Omron Sysmac Studio project testbed_1 (Sysmac Studio 1.30.0.17, StandardProject)

# Controller testbed_1: NX102-1000 version 1.40
Units and slaves: Unit 1 : NX-ECS112 (N1); Unit 2 : NX-PF0730 (N2); Unit 3 : NX-OD5256 (N3); Unit 4 : NX-ID5442 (N4); Unit 5 : NX-AD2604 (N5)
Axis Ax_Servo, settings changed from default: AxisType=ServoType, UnitsConversion=EnumElement5, UnitsNumerator=8388608, ReducerUse=EnumElement2, UnitsDenominator=360, TravelDistancePerWorkRotation=360, MotorGearRatio=30, MaxVelocity=600, MaxJogVelocity=90, InPositionBand=0.1, ZeroPositionBand=0.1, SoftwareLimitMode=ValidForSpecifiedValueDecreaseStop, PositiveSoftwareLimit=91, NegativeSoftwareLimit=-91, HomingVelocity=10, HomingApproachVelocity=10, CompensationVelocity=10, ModuloMAXPosition=180, ModuloMINPosition=-180
Axis Ax_Pendulum, settings changed from default: AxisNumber=1, AxisType=EncoderType, UnitsConversion=EnumElement5, UnitsNumerator=16384, UnitsDenominator=360, ActualVelocityFilterTime=100, CountMode=EnumElement2, ModuloMAXPosition=180, ModuloMINPosition=-180, EncoderTypes=Abs
Task PrimaryTask (priority 4, period or condition 1000): main

VAR_GLOBAL
    N1_Ch1_Encoder_Present_Position : DINT;  (* at IOBus://unit#1/Ch1 Encoder Present Position *)
    N3_Output_Bit_00 : BOOL;  (* at IOBus://unit#3/Output Bit 16 bits/Output Bit 00 *)
    N3_Output_Bit_01 : BOOL;  (* at IOBus://unit#3/Output Bit 16 bits/Output Bit 01 *)
    N3_Output_Bit_02 : BOOL;  (* at IOBus://unit#3/Output Bit 16 bits/Output Bit 02 *)
    N3_Output_Bit_03 : BOOL;  (* at IOBus://unit#3/Output Bit 16 bits/Output Bit 03 *)
    N4_Input_Bit_00 : BOOL;  (* at IOBus://unit#4/Input Bit 16 bits/Input Bit 00 *)
    N4_Input_Bit_01 : BOOL;  (* at IOBus://unit#4/Input Bit 16 bits/Input Bit 01 *)
    N4_Input_Bit_02 : BOOL;  (* at IOBus://unit#4/Input Bit 16 bits/Input Bit 02 *)
    N5_Ch1_Analog_Input_Value : INT;  (* at IOBus://unit#5/Ch1 Analog Input Value; published *)
END_VAR
VAR_GLOBAL CONSTANT
    Ax_Servo : _sAXIS_REF;  (* at MC://_MC_AX[0] *)
    Ax_Pendulum : _sAXIS_REF;  (* at MC://_MC_AX[1] *)
END_VAR
VAR_GLOBAL
    P0_System_State : UINT := 0;  (* published *)
    P0_Activate_Brake : BOOL := False;  (* published *)
    P0_Activate_Clutch : BOOL := False;  (* published *)
END_VAR
VAR_GLOBAL CONSTANT
    P0_SSI_Encoder_Offset : INT := 7822;  (* published *)
END_VAR
VAR_GLOBAL
    P0_SSI_Encoder_Degree_Position : LREAL := 0.0;  (* published *)
    P1_Enable : BOOL := False;  (* published *)
    P1_Upper_Position : LREAL := -60;  (* published *)
    P1_Start_Experiment : BOOL := False;  (* published *)
    P2_Enable : BOOL := False;  (* published *)
    P2_Start_Experiment : BOOL := False;  (* published *)
    P2_Displacement_Amplitude : LREAL := 10.0;  (* published *)
    P2_Frequency : LREAL := 0.1;  (* published *)
    P2_Cycles : UINT := 2;  (* published *)
    P3_Enable : BOOL := False;  (* published *)
    P3_Start_Experiment : BOOL := False;  (* published *)
    P3_Torque_Amplitude : LREAL := 2.0;  (* published *)
    P3_Frequency : LREAL := 0.1;  (* published *)
    P3_Cycles : UINT := 2;  (* published *)
    P0_Terminate : BOOL := False;  (* published *)
    P0_Relaxed_Position : LREAL := -5.0;  (* published *)
    P4_Start_Experiment : BOOL := False;  (* published *)
    P4_Displacement_Ramp_Slope : LREAL := 1.0;  (* published *)
    P5_Start_Experiment : BOOL := False;  (* published *)
    P4_Enable : BOOL := False;  (* published *)
    P5_Enable : BOOL := False;  (* published *)
    P5_Torque_Ramp_Slope : LREAL := 1.0;  (* published *)
    P5_Max_Torque : LREAL := 300.0;  (* published *)
    P0_Analog_Torque : LREAL := 0.0;  (* published *)
END_VAR

PROGRAM main
VAR
    fbk_P0_Brake_On : TON;
    P1_Pendulum_Vel_Abs : LREAL;
    fbk_P0_Brake_Off : TON;
    fbk_P0_Clutch_On : TON;
    fbk_P0_Clutch_Off : TON;
    fbk_P0_Servo_Activation : MC_Power;
    P2_Experiment_Time : LREAL;
    P2_Sin_Arg : LREAL;
    P2_Target_Position : LREAL;
    fbk_P2_Move_Sinusoidally : MC_SyncMoveAbsolute;
    fbk_P1_Move_To_Upper_Position : MC_MoveAbsolute;
    P3_Experiment_Time : LREAL;
    P3_Target_Torque : LREAL;
    fbk_P3_Torque_Sinusoidally : MC_TorqueControl;
    P3_Sin_Arg : LREAL;
    P2_Start_Position : LREAL;
    fbk_P0_Sync_Servo_To_Pendulum : MC_SetPosition;
    P1_Counter_Reset : BOOL;
    fbk_P1_Speed_Change_Counter : CTU;
    P3_Torque_Control_Trigger : BOOL;
    fbk_P0_Sync_Servo_Home_Offset : MC_HomeWithParameter;
    P0_Homing_Parameters : _sHOMING_REF;
    fbk_P0_Limit_Torque : MC_SetTorqueLimit;
    P0_Max_Position : LREAL;
    P0_Next_Protocol_State : UINT;
    fbk_P4_Move_Slowly : MC_MoveVelocity;
    fbk_P5_Torque_Slowly : MC_TorqueControl;
    fbk_P2_Stop_Motion : MC_Stop;
    fbk_P3_Stop_Motion : MC_Stop;
    fbk_P4_Stop_Motion : MC_Stop;
    fbk_P5_Stop_Motion : MC_Stop;
END_VAR
VAR CONSTANT
    P0_Rated_Load_Torque : LREAL := 201.912;  (* 7.16 Nm * 30 * 0.94% *)
END_VAR
VAR
    P5_Max_Torque_Perc : LREAL;
    P5_Torque_Ramp_Slope_Perc : LREAL;
    P3_Target_Torque_Perc : LREAL;
    fbk_P1_Mantain_Position : MC_MoveAbsolute;
    fbk_P0_End_Maintain_Position : MC_MoveAbsolute;
    fbk_P0_Contact_Maintain_Position : MC_MoveAbsolute;
    fbk_P0_Contact_Move_To_Contact_Position : MC_MoveVelocity;
    fbk_P0_End_Move_To_Relaxed_Position : MC_MoveAbsolute;
    fbk_P0_Init_Delay_Set_Home : TON;
    fbk_P0_Init_Set_Home : MC_Home;
    P0_Contact_Detection_Counter : UINT;
END_VAR
VAR CONSTANT
    P0_Contact_Detection_Threshold : LREAL := 4.0;  (* 4.0 Nm *)
END_VAR
VAR
    fbk_P0_Contact_Stop_Motion : MC_Stop;
    P4_Detach_Detection_Counter : UINT;
    P5_Detach_Detection_Counter : UINT;
    fbk_P0_Contact_Delay : TON;
    fbk_P0_End_Stop_Motion : MC_Stop;
    fbk_P0_End_Delay : TON;
END_VAR
VAR_EXTERNAL CONSTANT
    Ax_Servo : _sAXIS_REF;
    Ax_Pendulum : _sAXIS_REF;
END_VAR
VAR_EXTERNAL
    P0_System_State : UINT;
    N1_Ch1_Encoder_Present_Position : DINT;
    N3_Output_Bit_00 : BOOL;  (* clutch *)
    N3_Output_Bit_01 : BOOL;  (* brake *)
    N5_Ch1_Analog_Input_Value : INT;
    P0_Activate_Brake : BOOL;
    P0_Activate_Clutch : BOOL;
    P0_SSI_Encoder_Degree_Position : LREAL;
END_VAR
VAR_EXTERNAL CONSTANT
    P0_SSI_Encoder_Offset : INT;
END_VAR
VAR_EXTERNAL
    P1_Enable : BOOL;
    P1_Upper_Position : LREAL;
    P1_Start_Experiment : BOOL;
    P2_Enable : BOOL;
    P2_Start_Experiment : BOOL;
    P2_Displacement_Amplitude : LREAL;
    P2_Frequency : LREAL;
    P2_Cycles : UINT;
    P3_Enable : BOOL;
    P3_Start_Experiment : BOOL;
    P3_Torque_Amplitude : LREAL;
    P3_Frequency : LREAL;
    P3_Cycles : UINT;
    N4_Input_Bit_00 : BOOL;  (* push button *)
    N4_Input_Bit_01 : BOOL;  (* gate in *)
    P0_Terminate : BOOL;
    P0_Relaxed_Position : LREAL;
    P4_Start_Experiment : BOOL;
    P4_Displacement_Ramp_Slope : LREAL;
    P5_Start_Experiment : BOOL;
    P4_Enable : BOOL;
    P5_Enable : BOOL;
    P5_Torque_Ramp_Slope : LREAL;
    P5_Max_Torque : LREAL;
    N4_Input_Bit_02 : BOOL;  (* gate out *)
    N3_Output_Bit_02 : BOOL;  (* gate in *)
    N3_Output_Bit_03 : BOOL;  (* gate out *)
    P0_Analog_Torque : LREAL;
END_VAR
VAR
    _p1 : BOOL;
    _p2 : BOOL;
    _p3 : BOOL;
    _e4 : R_TRIG;
    _e5 : R_TRIG;
    _p6 : BOOL;
    _p7 : BOOL;
    _p8 : BOOL;
    _p9 : BOOL;
    _p10 : BOOL;
    _p11 : BOOL;
    _p12 : BOOL;
END_VAR

(* Section p0_init: ladder, written here as Structured Text *)

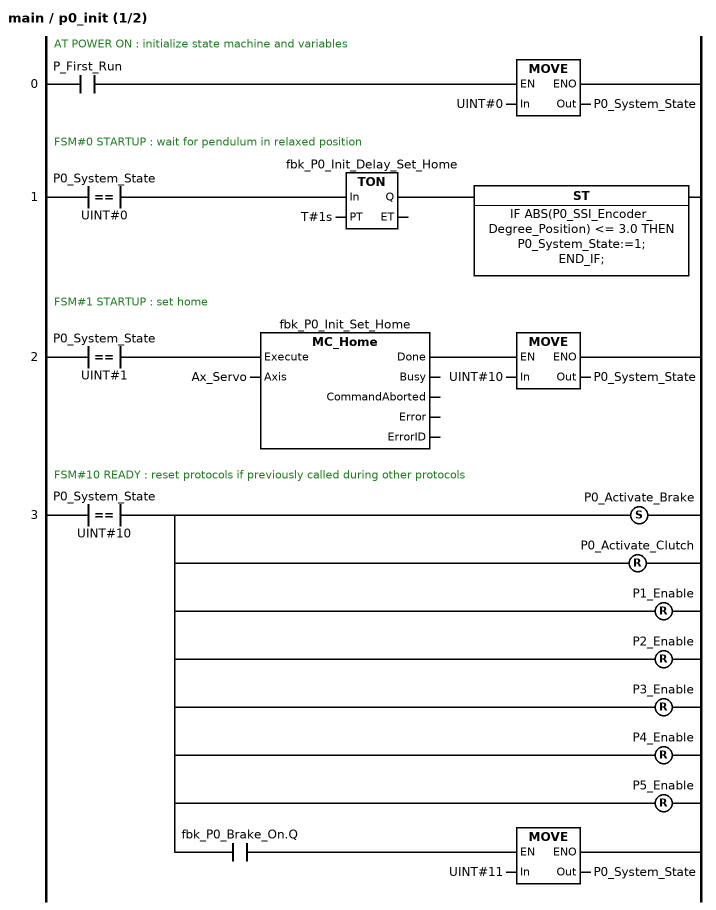
(* Rung 0: AT POWER ON : initialize state machine and variables *)
IF P_First_Run THEN P0_System_State := UINT#0; END_IF;
(* Rung 1: FSM#0 STARTUP : wait for pendulum in relaxed position *)
fbk_P0_Init_Delay_Set_Home(In := P0_System_State = UINT#0, PT := T#1s);
IF fbk_P0_Init_Delay_Set_Home.Q THEN
    IF ABS(P0_SSI_Encoder_Degree_Position) <= 3.0 THEN
    	P0_System_State:=1;
    END_IF;
END_IF;
(* Rung 2: FSM#1 STARTUP : set home *)
fbk_P0_Init_Set_Home(Execute := P0_System_State = UINT#1, Axis := Ax_Servo);
IF fbk_P0_Init_Set_Home.Done THEN P0_System_State := UINT#10; END_IF;
(* Rung 3: FSM#10 READY : reset protocols if previously called during other protocols *)
IF P0_System_State = UINT#10 THEN
    P0_Activate_Brake := TRUE;
    P0_Activate_Clutch := FALSE;
    P1_Enable := FALSE;
    P2_Enable := FALSE;
    P3_Enable := FALSE;
    P4_Enable := FALSE;
    P5_Enable := FALSE;
END_IF;
IF (P0_System_State = UINT#10) AND fbk_P0_Brake_On.Q THEN P0_System_State := UINT#11; END_IF;

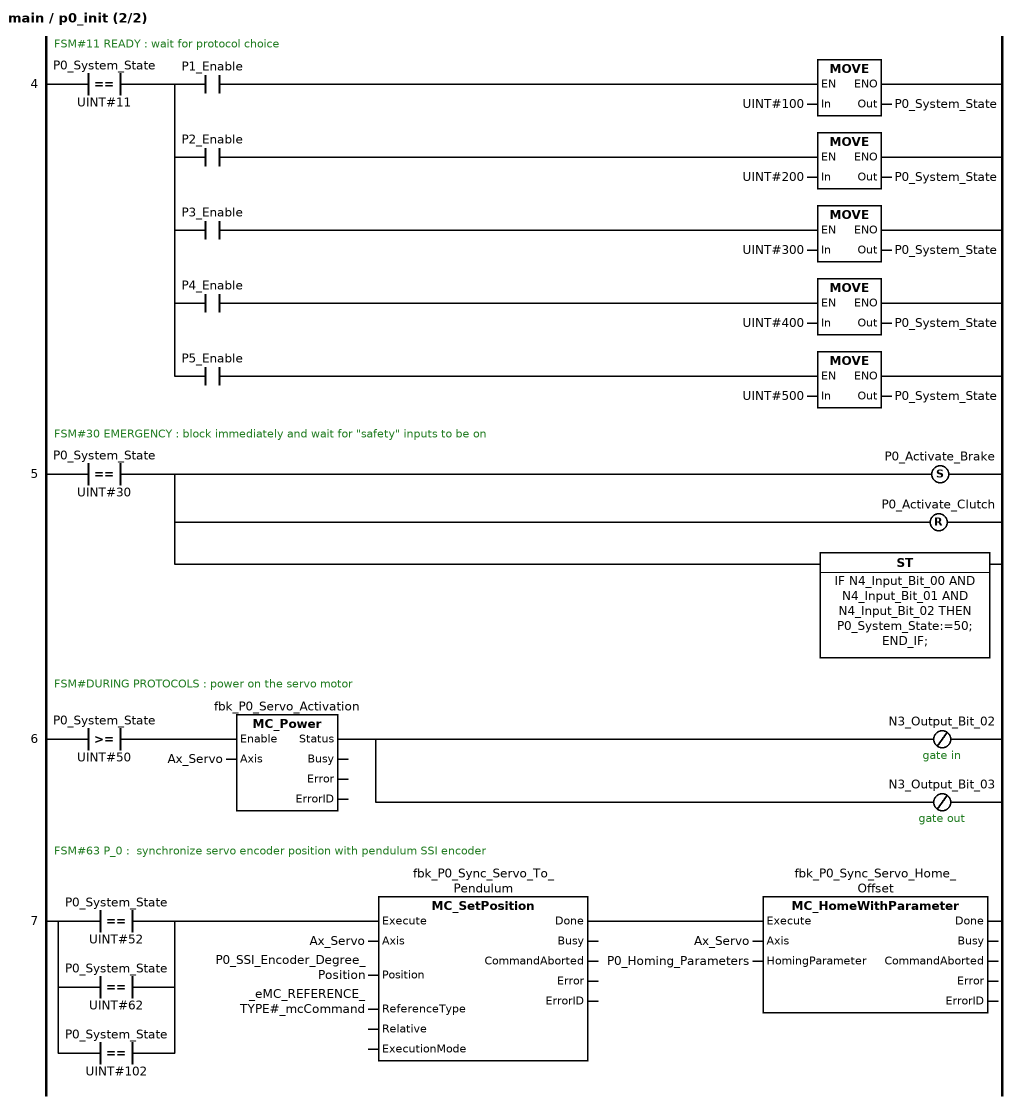
(* Rung 4: FSM#11 READY : wait for protocol choice *)
_p1 := P0_System_State = UINT#11;
IF (P0_System_State = UINT#11) AND P1_Enable THEN P0_System_State := UINT#100; END_IF;
IF _p1 AND P2_Enable THEN P0_System_State := UINT#200; END_IF;
IF _p1 AND P3_Enable THEN P0_System_State := UINT#300; END_IF;
IF _p1 AND P4_Enable THEN P0_System_State := UINT#400; END_IF;
IF _p1 AND P5_Enable THEN P0_System_State := UINT#500; END_IF;
(* Rung 5: FSM#30 EMERGENCY : block immediately and wait for "safety" inputs to be on *)
IF P0_System_State = UINT#30 THEN
    P0_Activate_Brake := TRUE;
    P0_Activate_Clutch := FALSE;
END_IF;
IF P0_System_State = UINT#30 THEN
    IF N4_Input_Bit_00 AND N4_Input_Bit_01 AND N4_Input_Bit_02 THEN
    	P0_System_State:=50;
    END_IF;
END_IF;
(* Rung 6: FSM#DURING PROTOCOLS : power on the servo motor *)
fbk_P0_Servo_Activation(Enable := P0_System_State >= UINT#50, Axis := Ax_Servo);
N3_Output_Bit_02 := NOT fbk_P0_Servo_Activation.Status;
N3_Output_Bit_03 := NOT fbk_P0_Servo_Activation.Status;
(* Rung 7: FSM#63 P_0 :  synchronize servo encoder position with pendulum SSI encoder *)
fbk_P0_Sync_Servo_To_Pendulum(Execute := (P0_System_State = UINT#52) OR (P0_System_State = UINT#62) OR (P0_System_State = UINT#102), Axis := Ax_Servo, Position := P0_SSI_Encoder_Degree_Position, ReferenceType := _eMC_REFERENCE_TYPE#_mcCommand);
fbk_P0_Sync_Servo_Home_Offset(Execute := fbk_P0_Sync_Servo_To_Pendulum.Done, Axis := Ax_Servo, HomingParameter := P0_Homing_Parameters);

(* Section p0_common: ladder, written here as Structured Text *)

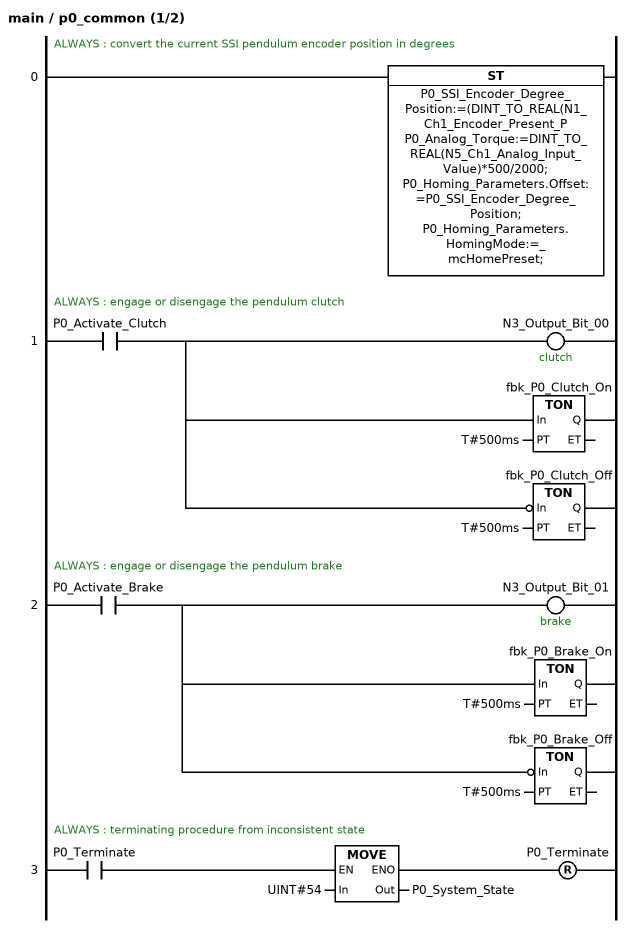
(* Rung 0: ALWAYS : convert the current SSI pendulum encoder position in degrees *)
P0_SSI_Encoder_Degree_Position:=(DINT_TO_REAL(N1_Ch1_Encoder_Present_Position-P0_SSI_Encoder_Offset)*360/16384);
P0_Analog_Torque:=DINT_TO_REAL(N5_Ch1_Analog_Input_Value)*500/2000;
P0_Homing_Parameters.Offset:=P0_SSI_Encoder_Degree_Position;
P0_Homing_Parameters.HomingMode:=_mcHomePreset;
(* Rung 1: ALWAYS : engage or disengage the pendulum clutch *)
N3_Output_Bit_00 := P0_Activate_Clutch;
fbk_P0_Clutch_On(In := P0_Activate_Clutch, PT := T#500ms);
fbk_P0_Clutch_Off(In := NOT P0_Activate_Clutch, PT := T#500ms);
(* Rung 2: ALWAYS : engage or disengage the pendulum brake *)
N3_Output_Bit_01 := P0_Activate_Brake;
fbk_P0_Brake_On(In := P0_Activate_Brake, PT := T#500ms);
fbk_P0_Brake_Off(In := NOT P0_Activate_Brake, PT := T#500ms);
(* Rung 3: ALWAYS : terminating procedure from inconsistent state *)
IF P0_Terminate THEN
    P0_System_State := UINT#54;
    P0_Terminate := FALSE;
END_IF;

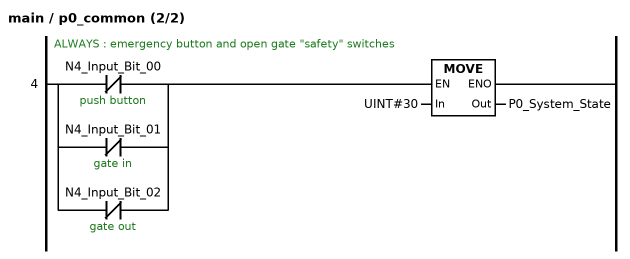
(* Rung 4: ALWAYS : emergency button and open gate "safety" switches *)
IF NOT N4_Input_Bit_00 OR NOT N4_Input_Bit_01 OR NOT N4_Input_Bit_02 THEN
    P0_System_State := UINT#30;
END_IF;

(* Section p0_end: ladder, written here as Structured Text *)

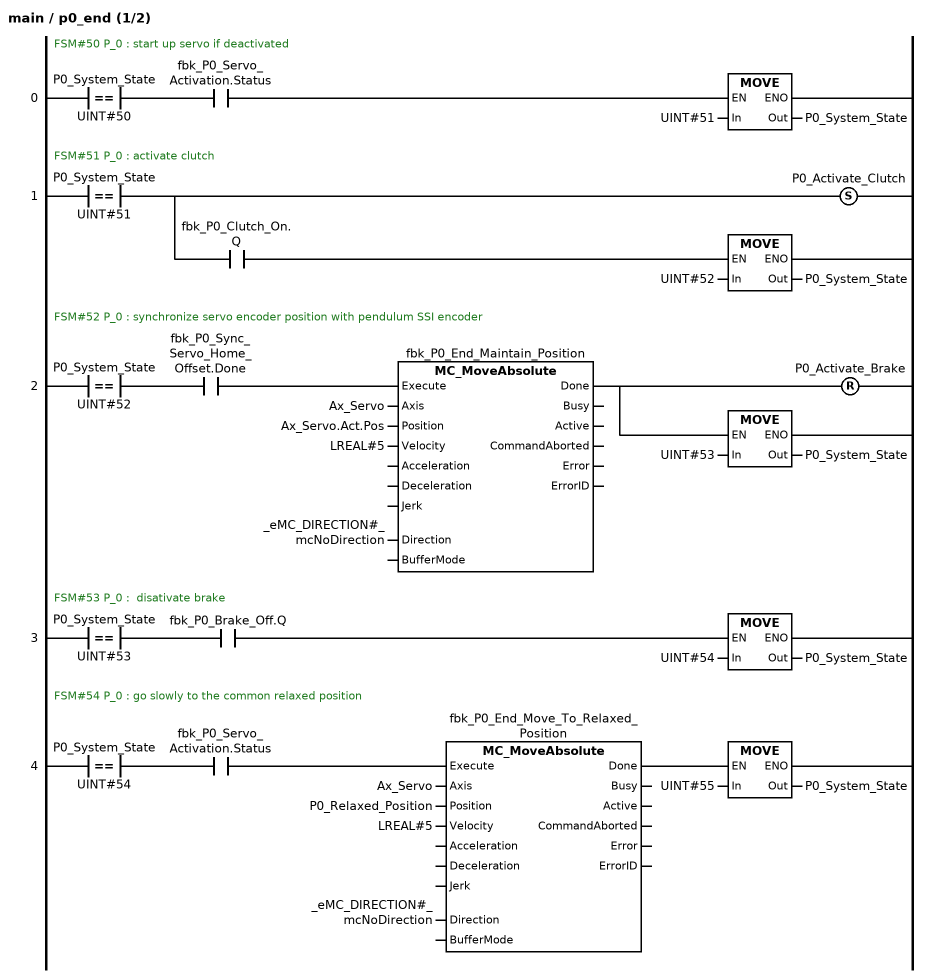
(* Rung 0: FSM#50 P_0 : start up servo if deactivated *)
IF (P0_System_State = UINT#50) AND fbk_P0_Servo_Activation.Status THEN P0_System_State := UINT#51; END_IF;
(* Rung 1: FSM#51 P_0 : activate clutch *)
IF P0_System_State = UINT#51 THEN P0_Activate_Clutch := TRUE; END_IF;
IF (P0_System_State = UINT#51) AND fbk_P0_Clutch_On.Q THEN P0_System_State := UINT#52; END_IF;
(* Rung 2: FSM#52 P_0 : synchronize servo encoder position with pendulum SSI encoder *)
fbk_P0_End_Maintain_Position(Execute := (P0_System_State = UINT#52) AND fbk_P0_Sync_Servo_Home_Offset.Done, Axis := Ax_Servo, Position := Ax_Servo.Act.Pos, Velocity := LREAL#5, Direction := _eMC_DIRECTION#_mcNoDirection);
IF fbk_P0_End_Maintain_Position.Done THEN
    P0_Activate_Brake := FALSE;
    P0_System_State := UINT#53;
END_IF;
(* Rung 3: FSM#53 P_0 :  disativate brake *)
IF (P0_System_State = UINT#53) AND fbk_P0_Brake_Off.Q THEN P0_System_State := UINT#54; END_IF;
(* Rung 4: FSM#54 P_0 : go slowly to the common relaxed position *)
fbk_P0_End_Move_To_Relaxed_Position(Execute := (P0_System_State = UINT#54) AND fbk_P0_Servo_Activation.Status, Axis := Ax_Servo, Position := P0_Relaxed_Position, Velocity := LREAL#5, Direction := _eMC_DIRECTION#_mcNoDirection);
IF fbk_P0_End_Move_To_Relaxed_Position.Done THEN P0_System_State := UINT#55; END_IF;

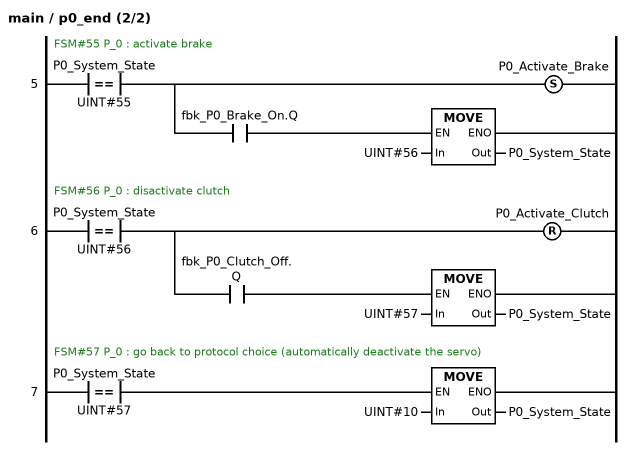
(* Rung 5: FSM#55 P_0 : activate brake *)
IF P0_System_State = UINT#55 THEN P0_Activate_Brake := TRUE; END_IF;
IF (P0_System_State = UINT#55) AND fbk_P0_Brake_On.Q THEN P0_System_State := UINT#56; END_IF;
(* Rung 6: FSM#56 P_0 : disactivate clutch *)
IF P0_System_State = UINT#56 THEN P0_Activate_Clutch := FALSE; END_IF;
IF (P0_System_State = UINT#56) AND fbk_P0_Clutch_Off.Q THEN P0_System_State := UINT#57; END_IF;
(* Rung 7: FSM#57 P_0 : go back to protocol choice (automatically deactivate the servo) *)
IF P0_System_State = UINT#57 THEN P0_System_State := UINT#10; END_IF;

(* Section p0_contact: ladder, written here as Structured Text *)

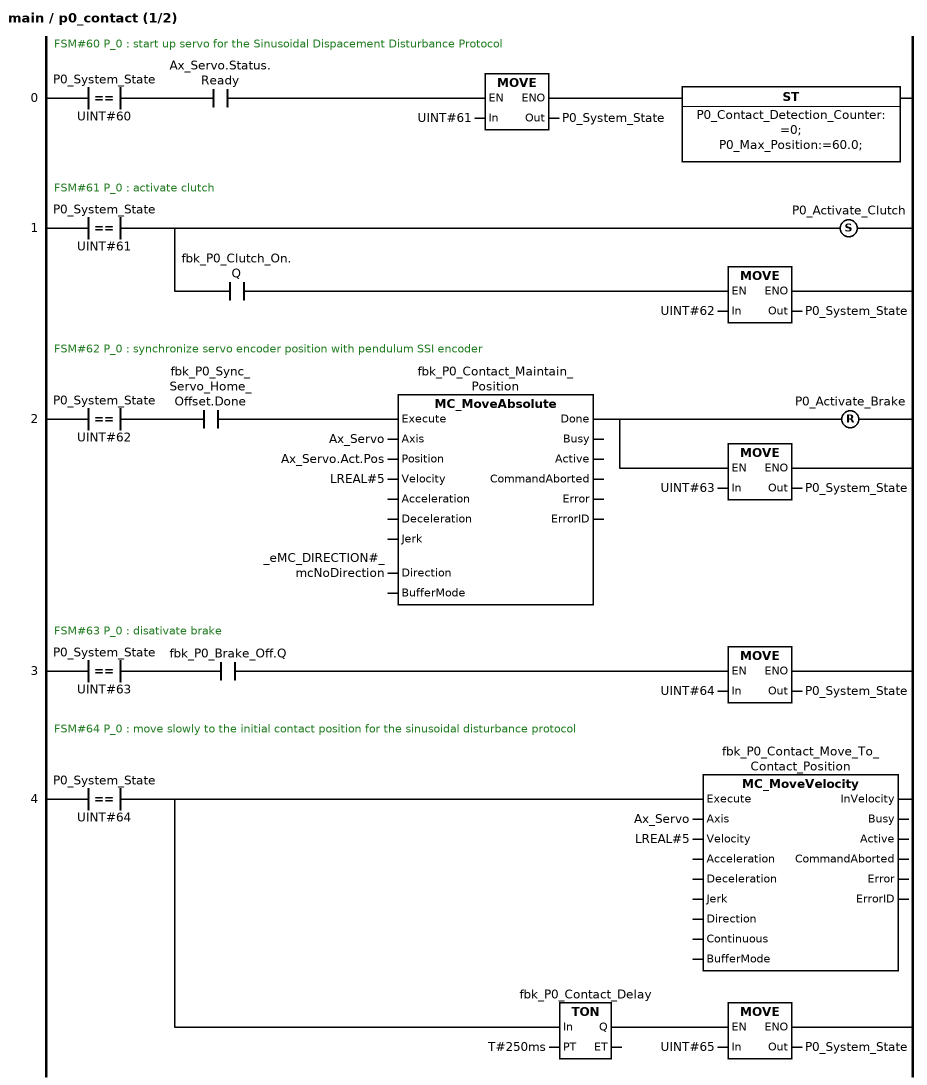
(* Rung 0: FSM#60 P_0 : start up servo for the Sinusoidal Dispacement Disturbance Protocol *)
_p2 := (P0_System_State = UINT#60) AND Ax_Servo.Status.Ready;
IF _p2 THEN P0_System_State := UINT#61; END_IF;
IF _p2 THEN
    P0_Contact_Detection_Counter:=0;
    P0_Max_Position:=60.0;
END_IF;
(* Rung 1: FSM#61 P_0 : activate clutch *)
IF P0_System_State = UINT#61 THEN P0_Activate_Clutch := TRUE; END_IF;
IF (P0_System_State = UINT#61) AND fbk_P0_Clutch_On.Q THEN P0_System_State := UINT#62; END_IF;
(* Rung 2: FSM#62 P_0 : synchronize servo encoder position with pendulum SSI encoder *)
fbk_P0_Contact_Maintain_Position(Execute := (P0_System_State = UINT#62) AND fbk_P0_Sync_Servo_Home_Offset.Done, Axis := Ax_Servo, Position := Ax_Servo.Act.Pos, Velocity := LREAL#5, Direction := _eMC_DIRECTION#_mcNoDirection);
IF fbk_P0_Contact_Maintain_Position.Done THEN
    P0_Activate_Brake := FALSE;
    P0_System_State := UINT#63;
END_IF;
(* Rung 3: FSM#63 P_0 : disativate brake *)
IF (P0_System_State = UINT#63) AND fbk_P0_Brake_Off.Q THEN P0_System_State := UINT#64; END_IF;
(* Rung 4: FSM#64 P_0 : move slowly to the initial contact position for the sinusoidal disturbance protocol *)
fbk_P0_Contact_Move_To_Contact_Position(Execute := P0_System_State = UINT#64, Axis := Ax_Servo, Velocity := LREAL#5);
fbk_P0_Contact_Delay(In := P0_System_State = UINT#64, PT := T#250ms);
IF fbk_P0_Contact_Delay.Q THEN P0_System_State := UINT#65; END_IF;

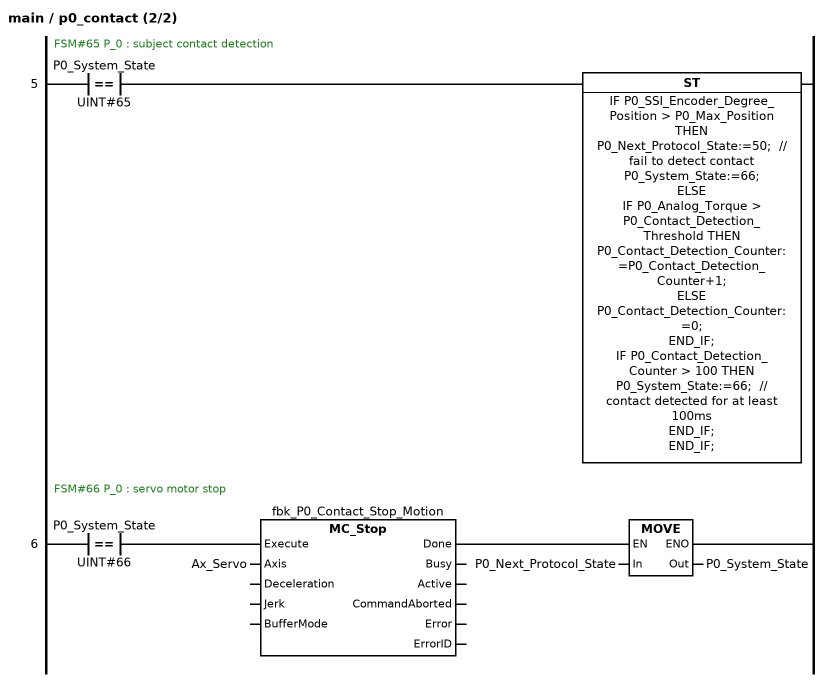
(* Rung 5: FSM#65 P_0 : subject contact detection *)
IF P0_System_State = UINT#65 THEN
    IF P0_SSI_Encoder_Degree_Position > P0_Max_Position THEN
    	P0_Next_Protocol_State:=50;  // fail to detect contact
    	P0_System_State:=66;
    ELSE
    	IF P0_Analog_Torque > P0_Contact_Detection_Threshold THEN
    		P0_Contact_Detection_Counter:=P0_Contact_Detection_Counter+1;
    	ELSE
    		P0_Contact_Detection_Counter:=0;
    	END_IF;
    
    	IF P0_Contact_Detection_Counter > 100 THEN
    		P0_System_State:=66;  // contact detected for at least 100ms
    	END_IF;
    END_IF;
END_IF;
(* Rung 6: FSM#66 P_0 : servo motor stop *)
fbk_P0_Contact_Stop_Motion(Execute := P0_System_State = UINT#66, Axis := Ax_Servo);
IF fbk_P0_Contact_Stop_Motion.Done THEN P0_System_State := P0_Next_Protocol_State; END_IF;

(* Section p1: ladder, written here as Structured Text *)

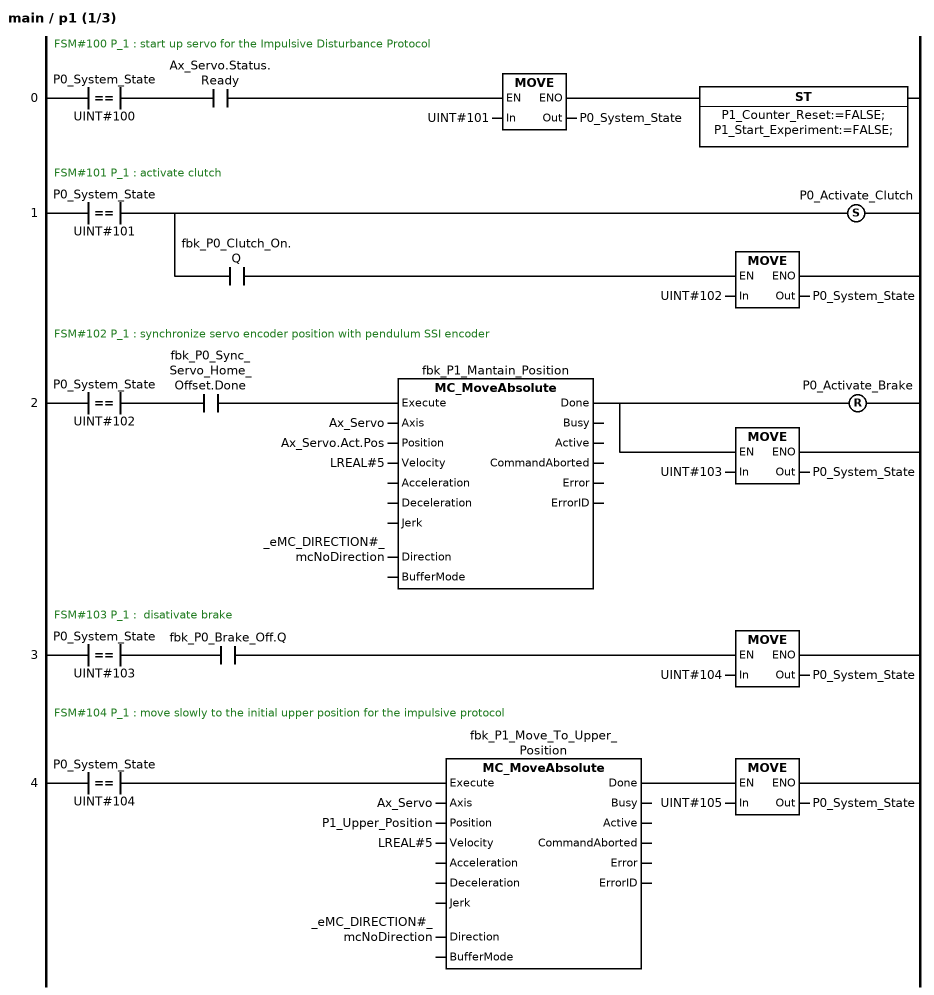
(* Rung 0: FSM#100 P_1 : start up servo for the Impulsive Disturbance Protocol *)
_p3 := (P0_System_State = UINT#100) AND Ax_Servo.Status.Ready;
IF _p3 THEN P0_System_State := UINT#101; END_IF;
IF _p3 THEN
    P1_Counter_Reset:=FALSE;
    P1_Start_Experiment:=FALSE;
END_IF;
(* Rung 1: FSM#101 P_1 : activate clutch *)
IF P0_System_State = UINT#101 THEN P0_Activate_Clutch := TRUE; END_IF;
IF (P0_System_State = UINT#101) AND fbk_P0_Clutch_On.Q THEN P0_System_State := UINT#102; END_IF;
(* Rung 2: FSM#102 P_1 : synchronize servo encoder position with pendulum SSI encoder *)
fbk_P1_Mantain_Position(Execute := (P0_System_State = UINT#102) AND fbk_P0_Sync_Servo_Home_Offset.Done, Axis := Ax_Servo, Position := Ax_Servo.Act.Pos, Velocity := LREAL#5, Direction := _eMC_DIRECTION#_mcNoDirection);
IF fbk_P1_Mantain_Position.Done THEN
    P0_Activate_Brake := FALSE;
    P0_System_State := UINT#103;
END_IF;
(* Rung 3: FSM#103 P_1 :  disativate brake *)
IF (P0_System_State = UINT#103) AND fbk_P0_Brake_Off.Q THEN P0_System_State := UINT#104; END_IF;
(* Rung 4: FSM#104 P_1 : move slowly to the initial upper position for the impulsive protocol *)
fbk_P1_Move_To_Upper_Position(Execute := P0_System_State = UINT#104, Axis := Ax_Servo, Position := P1_Upper_Position, Velocity := LREAL#5, Direction := _eMC_DIRECTION#_mcNoDirection);
IF fbk_P1_Move_To_Upper_Position.Done THEN P0_System_State := UINT#105; END_IF;

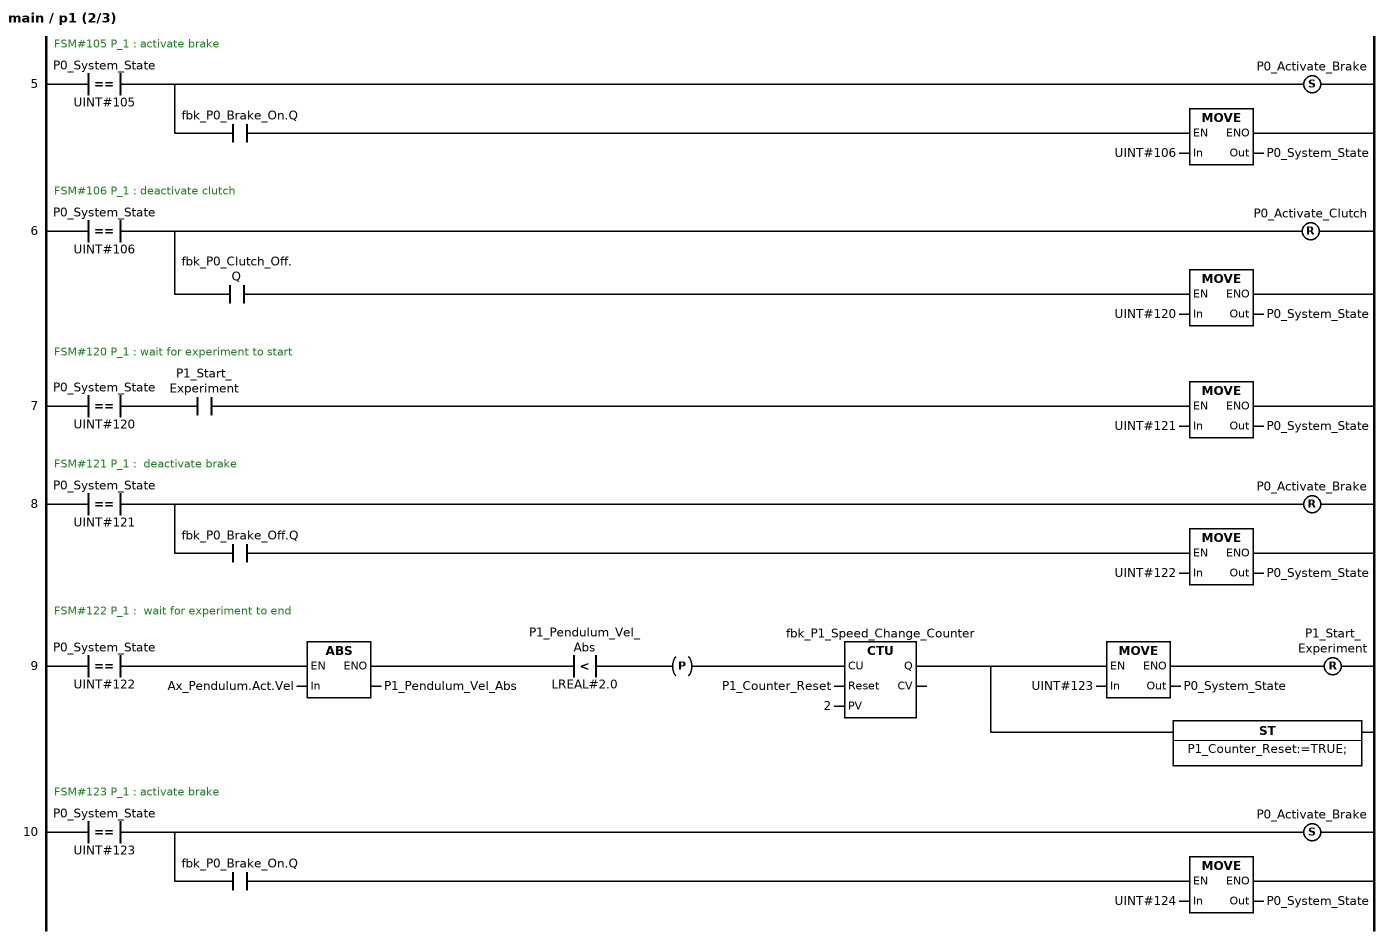
(* Rung 5: FSM#105 P_1 : activate brake *)
IF P0_System_State = UINT#105 THEN P0_Activate_Brake := TRUE; END_IF;
IF (P0_System_State = UINT#105) AND fbk_P0_Brake_On.Q THEN P0_System_State := UINT#106; END_IF;
(* Rung 6: FSM#106 P_1 : deactivate clutch *)
IF P0_System_State = UINT#106 THEN P0_Activate_Clutch := FALSE; END_IF;
IF (P0_System_State = UINT#106) AND fbk_P0_Clutch_Off.Q THEN P0_System_State := UINT#120; END_IF;
(* Rung 7: FSM#120 P_1 : wait for experiment to start *)
IF (P0_System_State = UINT#120) AND P1_Start_Experiment THEN P0_System_State := UINT#121; END_IF;
(* Rung 8: FSM#121 P_1 :  deactivate brake *)
IF P0_System_State = UINT#121 THEN P0_Activate_Brake := FALSE; END_IF;
IF (P0_System_State = UINT#121) AND fbk_P0_Brake_Off.Q THEN P0_System_State := UINT#122; END_IF;
(* Rung 9: FSM#122 P_1 :  wait for experiment to end *)
IF P0_System_State = UINT#122 THEN P1_Pendulum_Vel_Abs := ABS(In := Ax_Pendulum.Act.Vel); END_IF;
_e4(CLK := (P0_System_State = UINT#122) AND (P1_Pendulum_Vel_Abs < LREAL#2.0));
_e5(CLK := _e4.Q);
fbk_P1_Speed_Change_Counter(CU := _e5.Q, Reset := P1_Counter_Reset, PV := 2);
IF fbk_P1_Speed_Change_Counter.Q THEN
    P0_System_State := UINT#123;
    P1_Start_Experiment := FALSE;
END_IF;
IF fbk_P1_Speed_Change_Counter.Q THEN
    P1_Counter_Reset:=TRUE;
END_IF;
(* Rung 10: FSM#123 P_1 : activate brake *)
IF P0_System_State = UINT#123 THEN P0_Activate_Brake := TRUE; END_IF;
IF (P0_System_State = UINT#123) AND fbk_P0_Brake_On.Q THEN P0_System_State := UINT#124; END_IF;

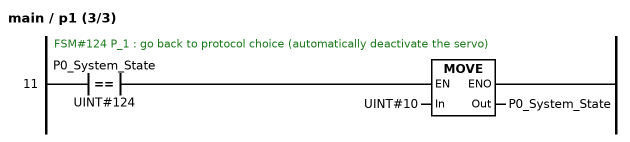
(* Rung 11: FSM#124 P_1 : go back to protocol choice (automatically deactivate the servo) *)
IF P0_System_State = UINT#124 THEN P0_System_State := UINT#10; END_IF;

(* Section p2: ladder, written here as Structured Text *)

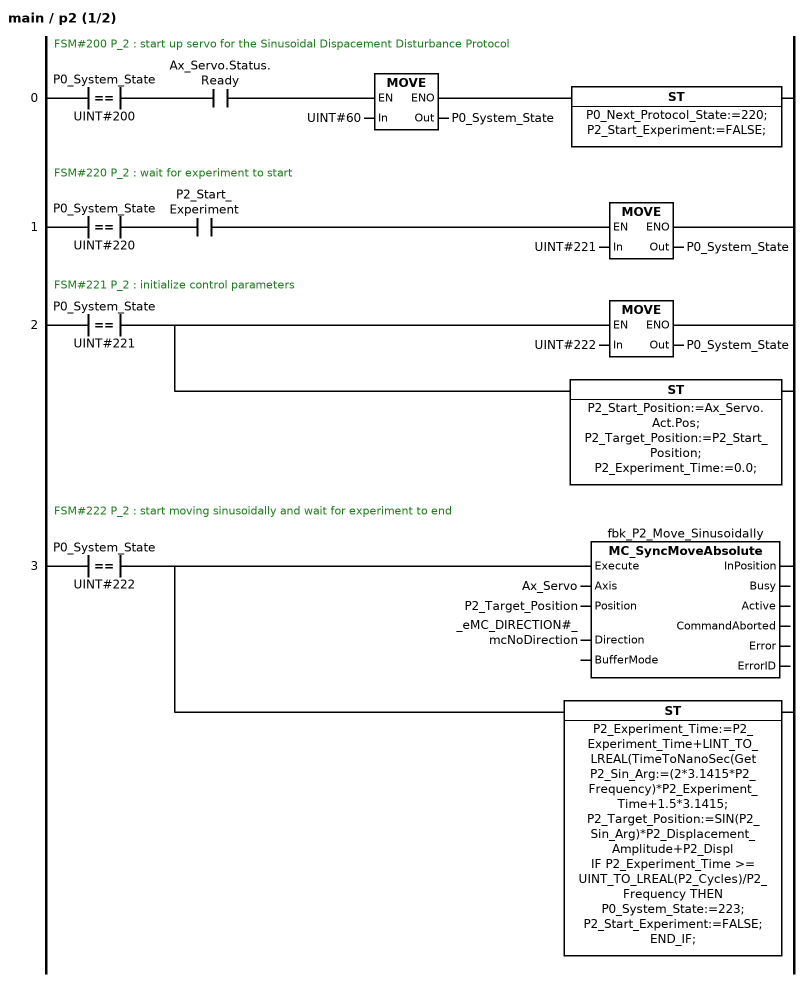
(* Rung 0: FSM#200 P_2 : start up servo for the Sinusoidal Dispacement Disturbance Protocol *)
_p6 := (P0_System_State = UINT#200) AND Ax_Servo.Status.Ready;
IF _p6 THEN P0_System_State := UINT#60; END_IF;
IF _p6 THEN
    P0_Next_Protocol_State:=220;
    P2_Start_Experiment:=FALSE;
END_IF;
(* Rung 1: FSM#220 P_2 : wait for experiment to start *)
IF (P0_System_State = UINT#220) AND P2_Start_Experiment THEN P0_System_State := UINT#221; END_IF;
(* Rung 2: FSM#221 P_2 : initialize control parameters *)
_p7 := P0_System_State = UINT#221;
IF _p7 THEN P0_System_State := UINT#222; END_IF;
IF _p7 THEN
    P2_Start_Position:=Ax_Servo.Act.Pos;
    P2_Target_Position:=P2_Start_Position;
    P2_Experiment_Time:=0.0;
END_IF;
(* Rung 3: FSM#222 P_2 : start moving sinusoidally and wait for experiment to end *)
fbk_P2_Move_Sinusoidally(Execute := P0_System_State = UINT#222, Axis := Ax_Servo, Position := P2_Target_Position, Direction := _eMC_DIRECTION#_mcNoDirection);
IF P0_System_State = UINT#222 THEN
    P2_Experiment_Time:=P2_Experiment_Time+LINT_TO_LREAL(TimeToNanoSec(GetMyTaskInterval()))/1000000000;
    
    P2_Sin_Arg:=(2*3.1415*P2_Frequency)*P2_Experiment_Time+1.5*3.1415;
    P2_Target_Position:=SIN(P2_Sin_Arg)*P2_Displacement_Amplitude+P2_Displacement_Amplitude+P2_Start_Position;
    
    IF P2_Experiment_Time >= UINT_TO_LREAL(P2_Cycles)/P2_Frequency THEN
    	P0_System_State:=223;
    	P2_Start_Experiment:=FALSE;
    END_IF;
END_IF;

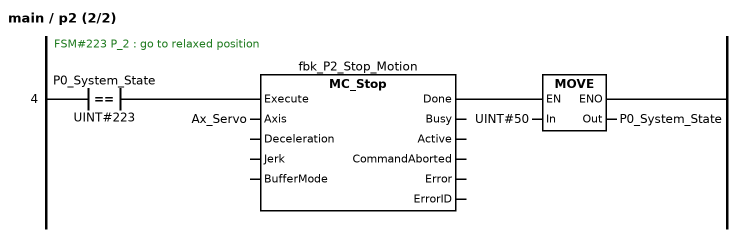
(* Rung 4: FSM#223 P_2 : go to relaxed position *)
fbk_P2_Stop_Motion(Execute := P0_System_State = UINT#223, Axis := Ax_Servo);
IF fbk_P2_Stop_Motion.Done THEN P0_System_State := UINT#50; END_IF;

(* Section p3: ladder, written here as Structured Text *)

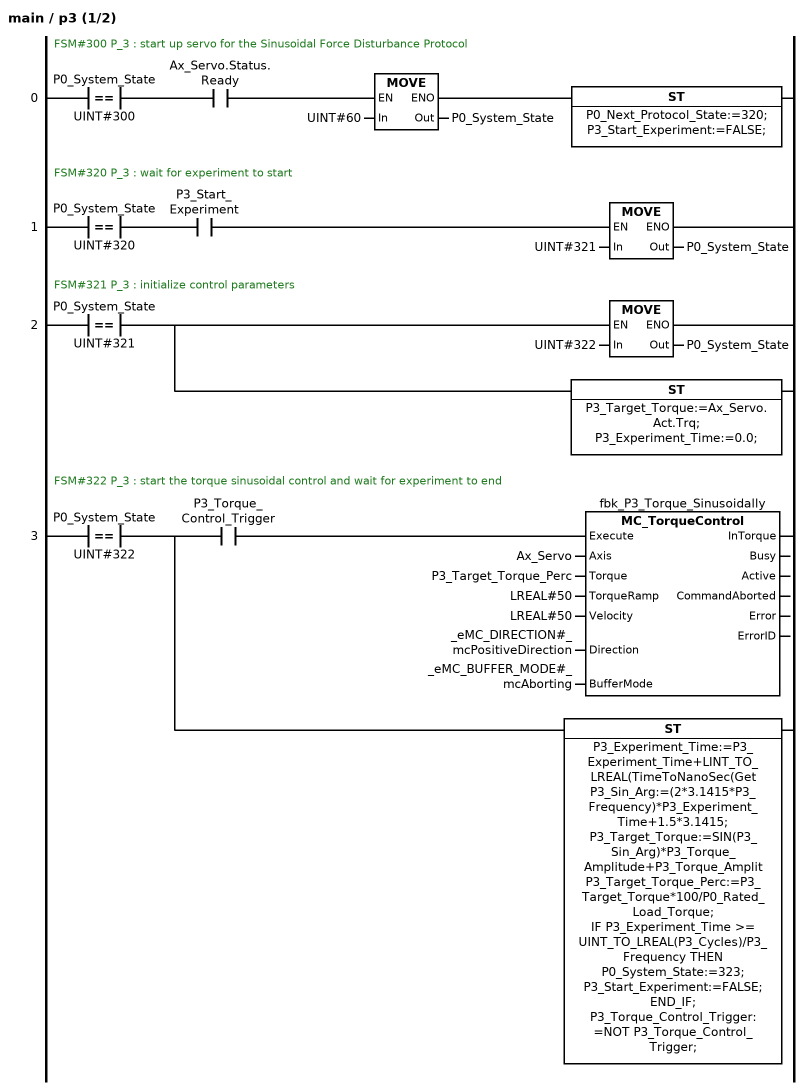
(* Rung 0: FSM#300 P_3 : start up servo for the Sinusoidal Force Disturbance Protocol *)
_p8 := (P0_System_State = UINT#300) AND Ax_Servo.Status.Ready;
IF _p8 THEN P0_System_State := UINT#60; END_IF;
IF _p8 THEN
    P0_Next_Protocol_State:=320;
    P3_Start_Experiment:=FALSE;
END_IF;
(* Rung 1: FSM#320 P_3 : wait for experiment to start *)
IF (P0_System_State = UINT#320) AND P3_Start_Experiment THEN P0_System_State := UINT#321; END_IF;
(* Rung 2: FSM#321 P_3 : initialize control parameters *)
_p9 := P0_System_State = UINT#321;
IF _p9 THEN P0_System_State := UINT#322; END_IF;
IF _p9 THEN
    P3_Target_Torque:=Ax_Servo.Act.Trq;
    P3_Experiment_Time:=0.0;
END_IF;
(* Rung 3: FSM#322 P_3 : start the torque sinusoidal control and wait for experiment to end *)
fbk_P3_Torque_Sinusoidally(Execute := (P0_System_State = UINT#322) AND P3_Torque_Control_Trigger, Axis := Ax_Servo, Torque := P3_Target_Torque_Perc, TorqueRamp := LREAL#50, Velocity := LREAL#50, Direction := _eMC_DIRECTION#_mcPositiveDirection, BufferMode := _eMC_BUFFER_MODE#_mcAborting);
IF P0_System_State = UINT#322 THEN
    P3_Experiment_Time:=P3_Experiment_Time+LINT_TO_LREAL(TimeToNanoSec(GetMyTaskInterval()))/1000000000;
    
    P3_Sin_Arg:=(2*3.1415*P3_Frequency)*P3_Experiment_Time+1.5*3.1415;
    P3_Target_Torque:=SIN(P3_Sin_Arg)*P3_Torque_Amplitude+P3_Torque_Amplitude;
    P3_Target_Torque_Perc:=P3_Target_Torque*100/P0_Rated_Load_Torque;
    
    IF P3_Experiment_Time >= UINT_TO_LREAL(P3_Cycles)/P3_Frequency THEN
    	P0_System_State:=323;
    	P3_Start_Experiment:=FALSE;
    END_IF;
    
    P3_Torque_Control_Trigger:=NOT P3_Torque_Control_Trigger;
END_IF;

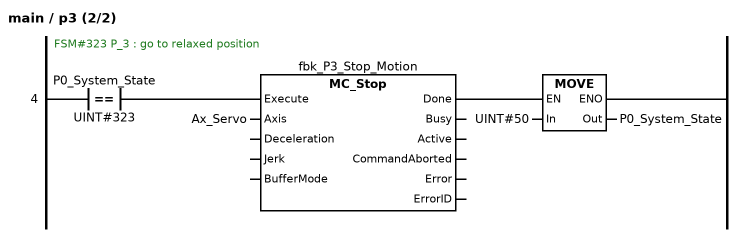
(* Rung 4: FSM#323 P_3 : go to relaxed position *)
fbk_P3_Stop_Motion(Execute := P0_System_State = UINT#323, Axis := Ax_Servo);
IF fbk_P3_Stop_Motion.Done THEN P0_System_State := UINT#50; END_IF;

(* Section p4: ladder, written here as Structured Text *)

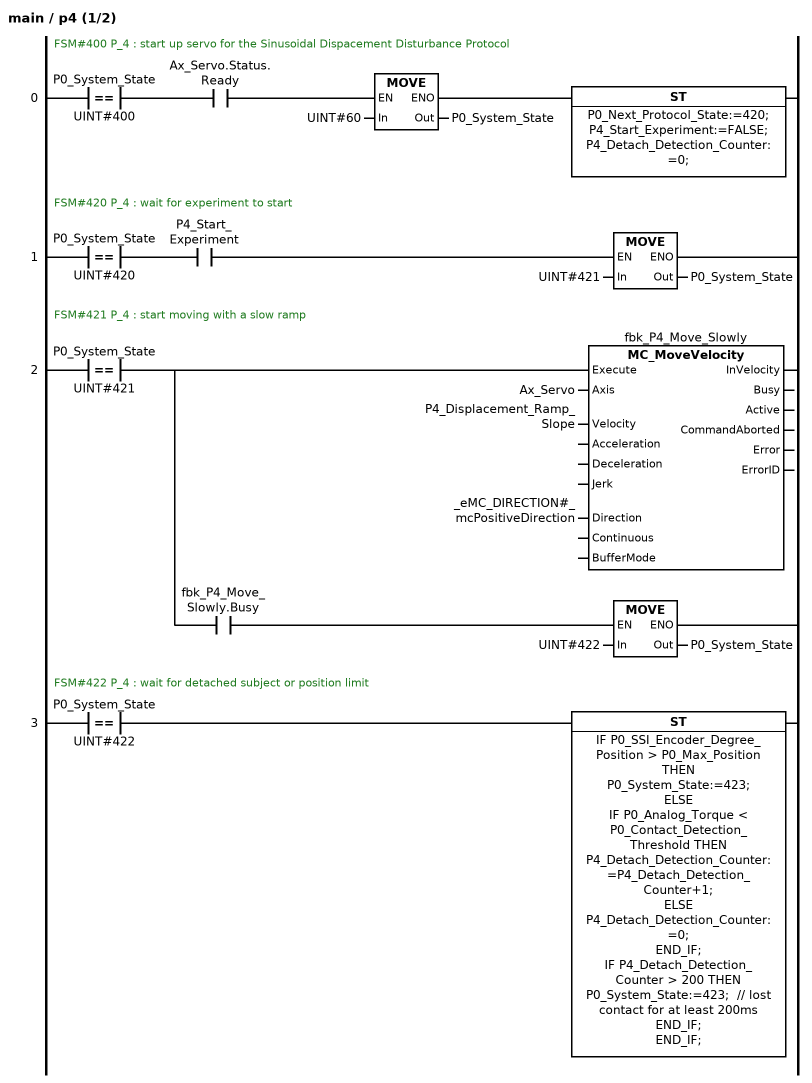
(* Rung 0: FSM#400 P_4 : start up servo for the Sinusoidal Dispacement Disturbance Protocol *)
_p10 := (P0_System_State = UINT#400) AND Ax_Servo.Status.Ready;
IF _p10 THEN P0_System_State := UINT#60; END_IF;
IF _p10 THEN
    P0_Next_Protocol_State:=420;
    P4_Start_Experiment:=FALSE;
    P4_Detach_Detection_Counter:=0;
END_IF;
(* Rung 1: FSM#420 P_4 : wait for experiment to start *)
IF (P0_System_State = UINT#420) AND P4_Start_Experiment THEN P0_System_State := UINT#421; END_IF;
(* Rung 2: FSM#421 P_4 : start moving with a slow ramp *)
fbk_P4_Move_Slowly(Execute := P0_System_State = UINT#421, Axis := Ax_Servo, Velocity := P4_Displacement_Ramp_Slope, Direction := _eMC_DIRECTION#_mcPositiveDirection);
IF (P0_System_State = UINT#421) AND fbk_P4_Move_Slowly.Busy THEN P0_System_State := UINT#422; END_IF;
(* Rung 3: FSM#422 P_4 : wait for detached subject or position limit *)
IF P0_System_State = UINT#422 THEN
    IF P0_SSI_Encoder_Degree_Position > P0_Max_Position THEN
    	P0_System_State:=423;
    ELSE
    	IF P0_Analog_Torque < P0_Contact_Detection_Threshold THEN
    		P4_Detach_Detection_Counter:=P4_Detach_Detection_Counter+1;
    	ELSE
    		P4_Detach_Detection_Counter:=0;
    	END_IF;
    
    	IF P4_Detach_Detection_Counter > 200 THEN
    		P0_System_State:=423;  // lost contact for at least 200ms
    	END_IF;
    END_IF;
END_IF;

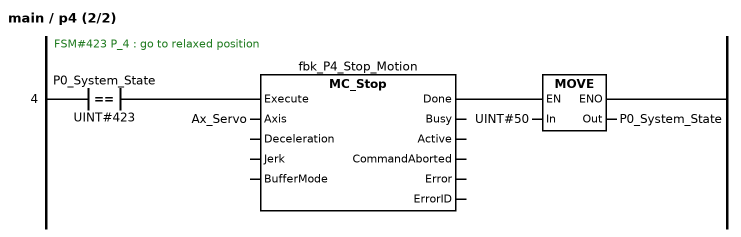
(* Rung 4: FSM#423 P_4 : go to relaxed position *)
fbk_P4_Stop_Motion(Execute := P0_System_State = UINT#423, Axis := Ax_Servo);
IF fbk_P4_Stop_Motion.Done THEN P0_System_State := UINT#50; END_IF;

(* Section p5: ladder, written here as Structured Text *)

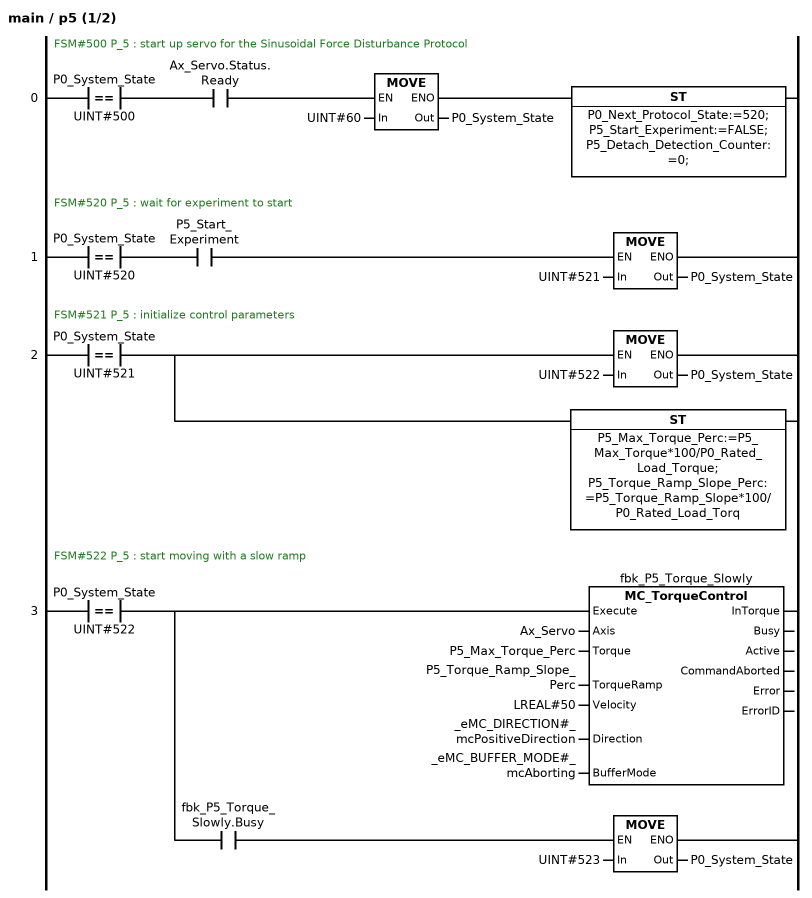
(* Rung 0: FSM#500 P_5 : start up servo for the Sinusoidal Force Disturbance Protocol *)
_p11 := (P0_System_State = UINT#500) AND Ax_Servo.Status.Ready;
IF _p11 THEN P0_System_State := UINT#60; END_IF;
IF _p11 THEN
    P0_Next_Protocol_State:=520;
    P5_Start_Experiment:=FALSE;
    P5_Detach_Detection_Counter:=0;
END_IF;
(* Rung 1: FSM#520 P_5 : wait for experiment to start *)
IF (P0_System_State = UINT#520) AND P5_Start_Experiment THEN P0_System_State := UINT#521; END_IF;
(* Rung 2: FSM#521 P_5 : initialize control parameters *)
_p12 := P0_System_State = UINT#521;
IF _p12 THEN P0_System_State := UINT#522; END_IF;
IF _p12 THEN
    P5_Max_Torque_Perc:=P5_Max_Torque*100/P0_Rated_Load_Torque;
    P5_Torque_Ramp_Slope_Perc:=P5_Torque_Ramp_Slope*100/P0_Rated_Load_Torque;
END_IF;
(* Rung 3: FSM#522 P_5 : start moving with a slow ramp *)
fbk_P5_Torque_Slowly(Execute := P0_System_State = UINT#522, Axis := Ax_Servo, Torque := P5_Max_Torque_Perc, TorqueRamp := P5_Torque_Ramp_Slope_Perc, Velocity := LREAL#50, Direction := _eMC_DIRECTION#_mcPositiveDirection, BufferMode := _eMC_BUFFER_MODE#_mcAborting);
IF (P0_System_State = UINT#522) AND fbk_P5_Torque_Slowly.Busy THEN P0_System_State := UINT#523; END_IF;

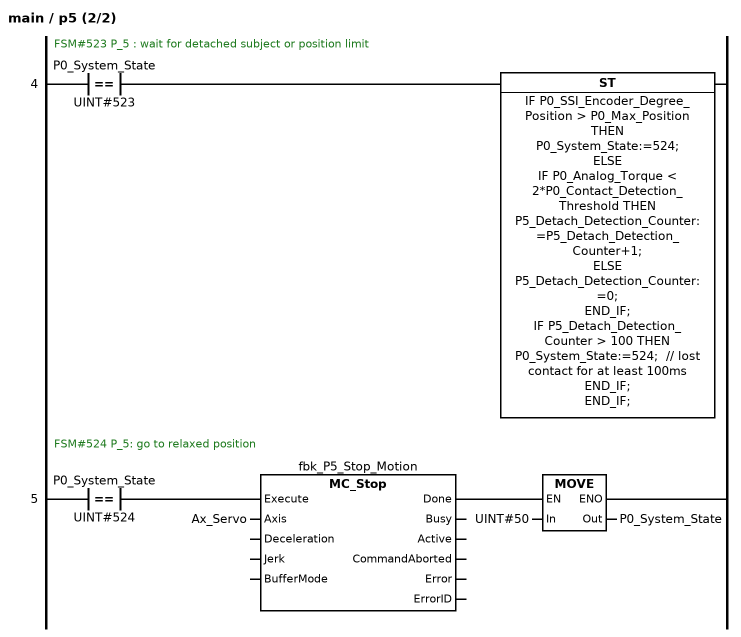
(* Rung 4: FSM#523 P_5 : wait for detached subject or position limit *)
IF P0_System_State = UINT#523 THEN
    IF P0_SSI_Encoder_Degree_Position > P0_Max_Position THEN
    	P0_System_State:=524;
    ELSE
    	IF P0_Analog_Torque < 2*P0_Contact_Detection_Threshold THEN
    		P5_Detach_Detection_Counter:=P5_Detach_Detection_Counter+1;
    	ELSE
    		P5_Detach_Detection_Counter:=0;
    	END_IF;
    
    	IF P5_Detach_Detection_Counter > 100 THEN
    		P0_System_State:=524;  // lost contact for at least 100ms
    	END_IF;
    END_IF;
END_IF;
(* Rung 5: FSM#524 P_5: go to relaxed position *)
fbk_P5_Stop_Motion(Execute := P0_System_State = UINT#524, Axis := Ax_Servo);
IF fbk_P5_Stop_Motion.Done THEN P0_System_State := UINT#50; END_IF;
END_PROGRAM